Yaskawa INFORM job: malben_program.JBI

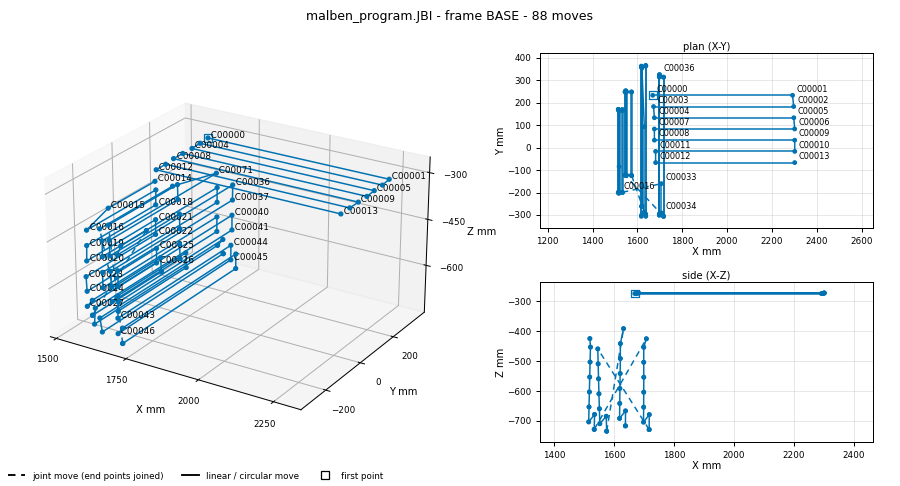
[picture p0: tool path of malben_program.JBI in frame BASE, 88 of 94 moves have a stored position in this frame; points joined in program order, loops and branches not executed]
/JOB
//NAME malben_program
//POS
///NPOS 88,0,88,0,0,0
///TOOL 0
///POSTYPE BASE
///RECTAN
///RCONF 0,0,0,0,0,0,0,0,0,0,0,0,0,0,0,0,0,0,0,0,0,0,0,0
C00000=1668.435673,233.475423,-274.172428,175.000000,5.000000,90.000000
C00001=2291.911749,233.475423,-274.172428,175.000000,5.000000,90.000000
C00002=2296.851748,183.475423,-274.026952,175.000000,5.000000,90.000000
C00003=1672.105793,183.475423,-274.026952,175.000000,5.000000,90.000000
C00004=1675.874125,133.475423,-273.500694,175.000000,5.000000,90.000000
C00005=2297.540153,133.475423,-273.500694,175.000000,5.000000,90.000000
C00006=2301.259379,83.475423,-272.802846,175.000000,5.000000,90.000000
C00007=1675.841540,83.475423,-272.802846,175.000000,5.000000,90.000000
C00008=1675.974173,33.475423,-272.491259,175.000000,5.000000,90.000000
C00009=2301.433775,33.475423,-272.491259,175.000000,5.000000,90.000000
C00010=2301.807350,-16.524577,-272.173336,175.000000,5.000000,90.000000
C00011=1681.303351,-16.524577,-272.173336,175.000000,5.000000,90.000000
C00012=1681.432312,-66.524577,-272.518020,175.000000,5.000000,90.000000
C00013=2301.497109,-66.524577,-272.518020,175.000000,5.000000,90.000000
C00014=1518.479294,164.562697,-424.700303,175.000000,-89.999999,5.000000
C00015=1518.479294,-84.458481,-424.700303,175.000000,-89.999999,5.000000
C00016=1520.450686,-199.361883,-453.160157,175.000000,-89.999999,5.000000
C00017=1520.450686,165.583095,-453.160157,175.000000,-89.999999,5.000000
C00018=1519.143907,165.377715,-503.160157,175.000000,-89.999999,5.000000
C00019=1519.143907,-199.039777,-503.160157,175.000000,-89.999999,5.000000
C00020=1517.931234,-199.520425,-553.160157,175.000000,-89.999999,5.000000
C00021=1517.931234,165.473756,-553.160157,175.000000,-89.999999,5.000000
C00022=1516.801469,165.483804,-603.160157,175.000000,-89.999999,5.000000
C00023=1516.801469,-203.687273,-603.160157,175.000000,-89.999999,5.000000
C00024=1515.593847,-199.039777,-653.160157,175.000000,-89.999999,5.000000
C00025=1515.593847,171.042802,-653.160157,175.000000,-89.999999,5.000000
C00026=1514.655118,170.957843,-703.160157,175.000000,-89.999999,5.000000
C00027=1514.655118,-199.199943,-703.160157,175.000000,-89.999999,5.000000
C00028=1534.135277,-199.660053,-678.160157,180.000000,-60.000000,0.000000
C00029=1534.135277,165.357325,-678.160157,180.000000,-60.000000,0.000000
C00030=1532.986245,170.762215,-728.160157,180.000000,-60.000000,0.000000
C00031=1532.986245,-199.039777,-728.160157,180.000000,-60.000000,0.000000
C00032=1532.986245,-199.039777,-728.160157,180.000000,-60.000000,0.000000
C00033=1707.297637,-160.264427,-425.389826,175.000000,-89.999999,5.000000
C00034=1707.297637,-290.468050,-425.389826,175.000000,-89.999999,5.000000
C00035=1698.543491,-296.135005,-453.830470,175.000000,-89.999999,5.000000
C00036=1698.543491,326.086108,-453.830470,175.000000,-89.999999,5.000000
C00037=1698.455560,324.501169,-503.830470,175.000000,-89.999999,5.000000
C00038=1698.455560,-296.135464,-503.830470,175.000000,-89.999999,5.000000
C00039=1698.607409,-296.135464,-553.830470,175.000000,-89.999999,5.000000
C00040=1698.607409,321.328537,-553.830470,175.000000,-89.999999,5.000000
C00041=1698.454230,321.328766,-603.830470,175.000000,-89.999999,5.000000
C00042=1698.454230,-296.563652,-603.830470,175.000000,-89.999999,5.000000
C00043=1698.216383,-300.894182,-653.830470,175.000000,-89.999999,5.000000
C00044=1698.216383,315.296956,-653.830470,175.000000,-89.999999,5.000000
C00045=1697.716752,315.510591,-703.830470,175.000000,-89.999999,5.000000
C00046=1697.716752,-300.894641,-703.830470,175.000000,-89.999999,5.000000
C00047=1717.044103,-305.652901,-678.830470,180.000000,-60.000000,0.000000
C00048=1717.044103,314.453200,-678.830470,180.000000,-60.000000,0.000000
C00049=1716.556742,314.453659,-728.830470,180.000000,-60.000000,0.000000
C00050=1716.556742,-305.653360,-728.830470,180.000000,-60.000000,0.000000
C00051=1716.556742,-305.653360,-728.830470,180.000000,-60.000000,0.000000
C00052=1544.970081,-122.877861,-459.225948,175.000000,-89.999999,5.000000
C00053=1544.970081,248.736792,-459.225948,175.000000,-89.999999,5.000000
C00054=1546.130786,248.644593,-509.225948,175.000000,-89.999999,5.000000
C00055=1546.130786,-122.535956,-509.225948,175.000000,-89.999999,5.000000
C00056=1547.451939,-122.877861,-559.225948,175.000000,-89.999999,5.000000
C00057=1547.451939,253.655271,-559.225948,175.000000,-89.999999,5.000000
C00058=1548.795390,253.495105,-609.225948,175.000000,-89.999999,5.000000
C00059=1548.795390,-123.193762,-609.225948,175.000000,-89.999999,5.000000
C00060=1550.223228,-122.807530,-659.225948,175.000000,-89.999999,5.000000
C00061=1550.223228,248.420300,-659.225948,175.000000,-89.999999,5.000000
C00062=1551.709648,248.736792,-709.225948,175.000000,-89.999999,5.000000
C00063=1551.709648,-122.877861,-709.225948,175.000000,-89.999999,5.000000
C00064=1573.113283,-123.038028,-684.225948,180.000000,-60.000000,0.000000
C00065=1573.113283,248.607359,-684.225948,180.000000,-60.000000,0.000000
C00066=1574.571207,248.055936,-734.225948,180.000000,-60.000000,0.000000
C00067=1574.571207,-124.672497,-734.225948,180.000000,-60.000000,0.000000
C00068=1574.571207,-124.672497,-734.225948,180.000000,-60.000000,0.000000
C00069=1630.958714,-286.067254,-391.404958,175.000000,-89.999999,5.000000
C00070=1630.958714,93.431035,-391.404958,175.000000,-89.999999,5.000000
C00071=1620.366614,354.769035,-441.404958,175.000000,-89.999999,5.000000
C00072=1620.366614,-260.685280,-441.404958,175.000000,-89.999999,5.000000
C00073=1620.227750,-261.513203,-491.404958,175.000000,-89.999999,5.000000
C00074=1620.227750,358.998140,-491.404958,175.000000,-89.999999,5.000000
C00075=1619.718447,358.999058,-541.404958,175.000000,-89.999999,5.000000
C00076=1619.718447,-261.707333,-541.404958,175.000000,-89.999999,5.000000
C00077=1618.807965,-261.033154,-591.404958,175.000000,-89.999999,5.000000
C00078=1618.807965,358.999058,-591.404958,175.000000,-89.999999,5.000000
C00079=1618.344207,359.055966,-641.404958,175.000000,-89.999999,5.000000
C00080=1618.344207,-301.212178,-641.404958,175.000000,-89.999999,5.000000
C00081=1617.747460,-306.161355,-691.404958,175.000000,-89.999999,5.000000
C00082=1617.747460,363.889491,-691.404958,175.000000,-89.999999,5.000000
C00083=1637.623559,363.967052,-666.404958,180.000000,-60.000000,0.000000
C00084=1637.623559,-306.160896,-666.404958,180.000000,-60.000000,0.000000
C00085=1637.288530,-295.508049,-716.404958,180.000000,-60.000000,0.000000
C00086=1637.288530,366.296157,-716.404958,180.000000,-60.000000,0.000000
C00087=1637.288530,366.296157,-716.404958,180.000000,-60.000000,0.000000
///POSTYPE PULSE
///PULSE
EC00000=0
EC00001=0
EC00002=0
EC00003=0
EC00004=0
EC00005=0
EC00006=0
EC00007=0
EC00008=0
EC00009=0
EC00010=0
EC00011=0
EC00012=0
EC00013=0
EC00014=0
EC00015=0
EC00016=0
EC00017=0
EC00018=0
EC00019=0
EC00020=0
EC00021=0
EC00022=0
EC00023=0
EC00024=0
EC00025=0
EC00026=0
EC00027=0
EC00028=0
EC00029=0
EC00030=0
EC00031=0
EC00032=92160
EC00033=92160
EC00034=92160
EC00035=92160
EC00036=92160
EC00037=92160
EC00038=92160
EC00039=92160
EC00040=92160
EC00041=92160
EC00042=92160
EC00043=92160
EC00044=92160
EC00045=92160
EC00046=92160
EC00047=92160
EC00048=92160
EC00049=92160
EC00050=92160
EC00051=184320
EC00052=184320
EC00053=184320
EC00054=184320
EC00055=184320
EC00056=184320
EC00057=184320
EC00058=184320
EC00059=184320
EC00060=184320
EC00061=184320
EC00062=184320
EC00063=184320
EC00064=184320
EC00065=184320
EC00066=184320
EC00067=184320
EC00068=276480
EC00069=276480
EC00070=276480
EC00071=276480
EC00072=276480
EC00073=276480
EC00074=276480
EC00075=276480
EC00076=276480
EC00077=276480
EC00078=276480
EC00079=276480
EC00080=276480
EC00081=276480
EC00082=276480
EC00083=276480
EC00084=276480
EC00085=276480
EC00086=276480
EC00087=368640
//INST
///DATE 2023/01/23 14:42
///ATTR SC,RW,RJ
////FRAME BASE
///GROUP1 RB1,ST1
NOP
MOVJ P009 EX000 VJ=15.00
MOVJ C00000 EC00000 VJ=15.0
CALL JOB:SPYON
MOVL C00001 EC00001 V=150.0
MOVL C00002 EC00002 V=150.0
MOVL C00003 EC00003 V=150.0
MOVL C00004 EC00004 V=150.0
MOVL C00005 EC00005 V=150.0
MOVL C00006 EC00006 V=150.0
MOVL C00007 EC00007 V=150.0
MOVL C00008 EC00008 V=150.0
MOVL C00009 EC00009 V=150.0
MOVL C00010 EC00010 V=150.0
MOVL C00011 EC00011 V=150.0
MOVL C00012 EC00012 V=150.0
MOVL C00013 EC00013 V=150.0
CALL JOB:SPYOF
MOVJ P009 VJ=15.00
MOVJ C00014 EC00014 VJ=15.0
CALL JOB:SPYON
MOVL C00015 EC00015 V=150.0
MOVL C00016 EC00016 V=150.0
MOVL C00017 EC00017 V=150.0
MOVL C00018 EC00018 V=150.0
MOVL C00019 EC00019 V=150.0
MOVL C00020 EC00020 V=150.0
MOVL C00021 EC00021 V=150.0
MOVL C00022 EC00022 V=150.0
MOVL C00023 EC00023 V=150.0
MOVL C00024 EC00024 V=150.0
MOVL C00025 EC00025 V=150.0
MOVL C00026 EC00026 V=150.0
MOVL C00027 EC00027 V=150.0
MOVL C00028 EC00028 V=150.0
MOVL C00029 EC00029 V=150.0
MOVL C00030 EC00030 V=150.0
MOVL C00031 EC00031 V=150.0
CALL JOB:SPYOF
MOVJ P009 VJ=15.00
MOVL C00032 EC00032 V=150.0
MOVJ C00033 EC00033 VJ=15.0
CALL JOB:SPYON
MOVL C00034 EC00034 V=150.0
MOVL C00035 EC00035 V=150.0
MOVL C00036 EC00036 V=150.0
MOVL C00037 EC00037 V=150.0
MOVL C00038 EC00038 V=150.0
MOVL C00039 EC00039 V=150.0
MOVL C00040 EC00040 V=150.0
MOVL C00041 EC00041 V=150.0
MOVL C00042 EC00042 V=150.0
MOVL C00043 EC00043 V=150.0
MOVL C00044 EC00044 V=150.0
MOVL C00045 EC00045 V=150.0
MOVL C00046 EC00046 V=150.0
MOVL C00047 EC00047 V=150.0
MOVL C00048 EC00048 V=150.0
MOVL C00049 EC00049 V=150.0
MOVL C00050 EC00050 V=150.0
CALL JOB:SPYOF
MOVJ P009 VJ=15.00
MOVL C00051 EC00051 V=150.0
MOVJ C00052 EC00052 VJ=15.0
CALL JOB:SPYON
MOVL C00053 EC00053 V=150.0
MOVL C00054 EC00054 V=150.0
MOVL C00055 EC00055 V=150.0
MOVL C00056 EC00056 V=150.0
MOVL C00057 EC00057 V=150.0
MOVL C00058 EC00058 V=150.0
MOVL C00059 EC00059 V=150.0
MOVL C00060 EC00060 V=150.0
MOVL C00061 EC00061 V=150.0
MOVL C00062 EC00062 V=150.0
MOVL C00063 EC00063 V=150.0
MOVL C00064 EC00064 V=150.0
MOVL C00065 EC00065 V=150.0
MOVL C00066 EC00066 V=150.0
MOVL C00067 EC00067 V=150.0
CALL JOB:SPYOF
MOVJ P009 VJ=15.00
MOVL C00068 EC00068 V=150.0
MOVJ C00069 EC00069 VJ=15.0
CALL JOB:SPYON
MOVL C00070 EC00070 V=150.0
MOVL C00071 EC00071 V=150.0
MOVL C00072 EC00072 V=150.0
MOVL C00073 EC00073 V=150.0
MOVL C00074 EC00074 V=150.0
MOVL C00075 EC00075 V=150.0
MOVL C00076 EC00076 V=150.0
MOVL C00077 EC00077 V=150.0
MOVL C00078 EC00078 V=150.0
MOVL C00079 EC00079 V=150.0
MOVL C00080 EC00080 V=150.0
MOVL C00081 EC00081 V=150.0
MOVL C00082 EC00082 V=150.0
MOVL C00083 EC00083 V=150.0
MOVL C00084 EC00084 V=150.0
MOVL C00085 EC00085 V=150.0
MOVL C00086 EC00086 V=150.0
CALL JOB:SPYOF
MOVJ P009 VJ=15.00
MOVL C00087 EC00087 V=150.0
END
